// TIA Portal V21 export
VAR_GLOBAL   // PLC tag table "PallettizzatoreReciveAnalogici"
END_VAR
VAR_GLOBAL CONSTANT   // user constants
   K_SegnaleDaPallettizzatore_NumeroStrati : Int := 1;
END_VAR
